// TIA Portal project "ASANSÖÖÖÖÖÖÖR" (V16)

(* hardware
DEVICE "S7-1200 station_1"  S7-1200 Station
   slot 0: "Rack_0"  S7-1200 Rack  Rack  V1.0
   slot 1: "PLC_1"  CPU 1212C DC/DC/Rly  6ES7 212-1HE40-0XB0  V4.4
*)

// ===== PLC "PLC_1"  CPU 1212C DC/DC/Rly =====

VAR_GLOBAL   // PLC tag table "Default tag table"
   "Kat 1 set yukarı" AT %M0.0 : Bool;
   "Kat 3 start" AT %I0.2 : Bool;
   "Kat 2 start" AT %I0.1 : Bool;
   "Set 3" AT %M0.2 : Bool;
   "Sensör 2" AT %I0.0 : Bool;
   "Kat 2 set yukarı" AT %M0.1 : Bool;
   "Kat 1 start" AT %I0.4 : Bool;
   "Sensör 1" AT %I0.5 : Bool;
   "Kat 2 aşağı" AT %M0.4 : Bool;
   "Kat 3 start set" AT %Q0.3 : Bool;
   "Kat 2 start set" AT %Q0.4 : Bool;
   "Kat 1 start set" AT %Q0.5 : Bool;
   "Sensör 3" AT %I0.6 : Bool;
   "Motor Yukarı" AT %Q0.2 : Bool;
   "Motor aşağı" AT %Q0.1 : Bool;
   "Kat 3 aşağı" AT %M0.3 : Bool;
END_VAR

ORGANIZATION_BLOCK "Main"   // OB1, LAD, ProgramCycle
TITLE = "Main Program Sweep (Cycle)"
{ S7_Optimized_Access := 'TRUE' }
VERSION : 0.1
   VAR_INPUT
      Initial_Call : Bool;   // Initial call of this OB
      Remanence : Bool;   // =True, if remanent data are available
   END_VAR
BEGIN

REGION Network 1
   // Kat 1 yukarı
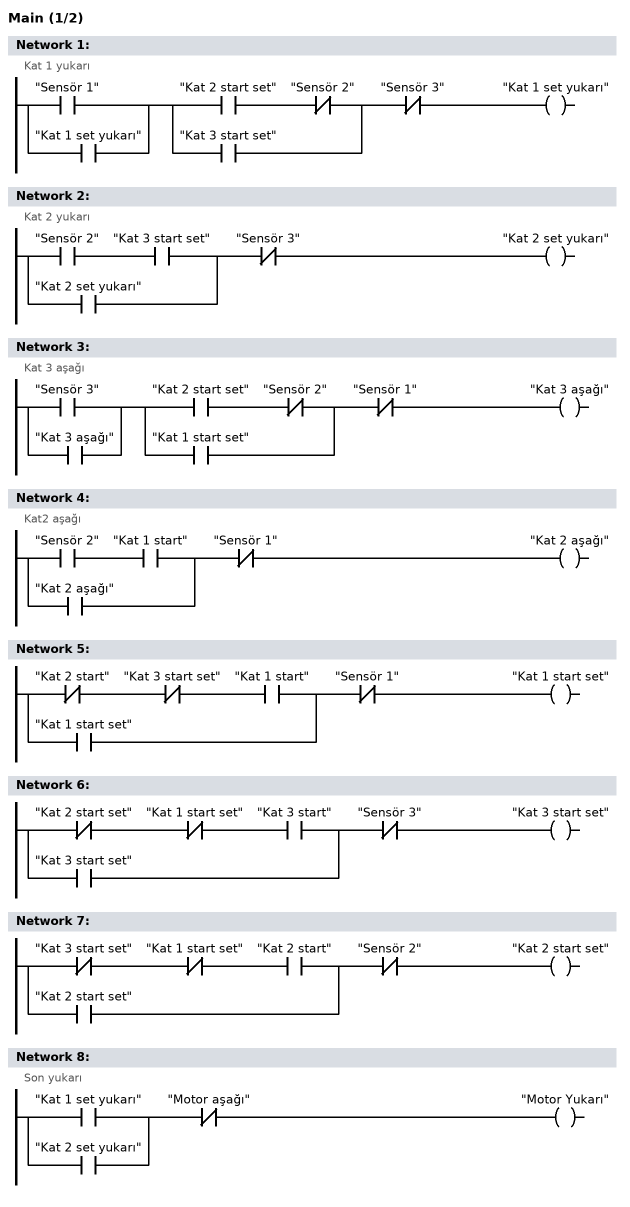
   RUNG wire#powerrail
      Contact( "Sensör 1" )
      wire#w1
      Contact( "Kat 2 start set" )
      I_Contact( "Sensör 2" )
      wire#w2
      I_Contact( "Sensör 3" )
      Coil( "Kat 1 set yukarı" )
   END_RUNG
   RUNG wire#powerrail
      Contact( "Kat 1 set yukarı" )
   END_RUNG wire#w1
   RUNG wire#w1
      Contact( "Kat 3 start set" )
   END_RUNG wire#w2
   // the same network as SCL:
   "Kat 1 set yukarı" := ("Sensör 1" OR "Kat 1 set yukarı") AND (("Kat 2 start set" AND NOT "Sensör 2") OR "Kat 3 start set") AND NOT "Sensör 3";
END_REGION

REGION Network 2
   // Kat 2 yukarı
   RUNG wire#powerrail
      Contact( "Sensör 2" )
      Contact( "Kat 3 start set" )
      wire#w1
      I_Contact( "Sensör 3" )
      Coil( "Kat 2 set yukarı" )
   END_RUNG
   RUNG wire#powerrail
      Contact( "Kat 2 set yukarı" )
   END_RUNG wire#w1
   // the same network as SCL:
   "Kat 2 set yukarı" := (("Sensör 2" AND "Kat 3 start set") OR "Kat 2 set yukarı") AND NOT "Sensör 3";
END_REGION

REGION Network 3
   // Kat 3 aşağı
   RUNG wire#powerrail
      Contact( "Sensör 3" )
      wire#w1
      Contact( "Kat 2 start set" )
      I_Contact( "Sensör 2" )
      wire#w2
      I_Contact( "Sensör 1" )
      Coil( "Kat 3 aşağı" )
   END_RUNG
   RUNG wire#powerrail
      Contact( "Kat 3 aşağı" )
   END_RUNG wire#w1
   RUNG wire#w1
      Contact( "Kat 1 start set" )
   END_RUNG wire#w2
   // the same network as SCL:
   "Kat 3 aşağı" := ("Sensör 3" OR "Kat 3 aşağı") AND (("Kat 2 start set" AND NOT "Sensör 2") OR "Kat 1 start set") AND NOT "Sensör 1";
END_REGION

REGION Network 4
   // Kat2 aşağı
   RUNG wire#powerrail
      Contact( "Sensör 2" )
      Contact( "Kat 1 start" )
      wire#w1
      I_Contact( "Sensör 1" )
      Coil( "Kat 2 aşağı" )
   END_RUNG
   RUNG wire#powerrail
      Contact( "Kat 2 aşağı" )
   END_RUNG wire#w1
   // the same network as SCL:
   "Kat 2 aşağı" := (("Sensör 2" AND "Kat 1 start") OR "Kat 2 aşağı") AND NOT "Sensör 1";
END_REGION

REGION Network 5
   RUNG wire#powerrail
      I_Contact( "Kat 2 start" )
      I_Contact( "Kat 3 start set" )
      Contact( "Kat 1 start" )
      wire#w1
      I_Contact( "Sensör 1" )
      Coil( "Kat 1 start set" )
   END_RUNG
   RUNG wire#powerrail
      Contact( "Kat 1 start set" )
   END_RUNG wire#w1
   // the same network as SCL:
   "Kat 1 start set" := ((NOT "Kat 2 start" AND NOT "Kat 3 start set" AND "Kat 1 start") OR "Kat 1 start set") AND NOT "Sensör 1";
END_REGION

REGION Network 6
   RUNG wire#powerrail
      I_Contact( "Kat 2 start set" )
      I_Contact( "Kat 1 start set" )
      Contact( "Kat 3 start" )
      wire#w1
      I_Contact( "Sensör 3" )
      Coil( "Kat 3 start set" )
   END_RUNG
   RUNG wire#powerrail
      Contact( "Kat 3 start set" )
   END_RUNG wire#w1
   // the same network as SCL:
   "Kat 3 start set" := ((NOT "Kat 2 start set" AND NOT "Kat 1 start set" AND "Kat 3 start") OR "Kat 3 start set") AND NOT "Sensör 3";
END_REGION

REGION Network 7
   RUNG wire#powerrail
      I_Contact( "Kat 3 start set" )
      I_Contact( "Kat 1 start set" )
      Contact( "Kat 2 start" )
      wire#w1
      I_Contact( "Sensör 2" )
      Coil( "Kat 2 start set" )
   END_RUNG
   RUNG wire#powerrail
      Contact( "Kat 2 start set" )
   END_RUNG wire#w1
   // the same network as SCL:
   "Kat 2 start set" := ((NOT "Kat 3 start set" AND NOT "Kat 1 start set" AND "Kat 2 start") OR "Kat 2 start set") AND NOT "Sensör 2";
END_REGION

REGION Network 8
   // Son yukarı
   RUNG wire#powerrail
      Contact( "Kat 1 set yukarı" )
      wire#w1
      I_Contact( "Motor aşağı" )
      Coil( "Motor Yukarı" )
   END_RUNG
   RUNG wire#powerrail
      Contact( "Kat 2 set yukarı" )
   END_RUNG wire#w1
   // the same network as SCL:
   "Motor Yukarı" := ("Kat 1 set yukarı" OR "Kat 2 set yukarı") AND NOT "Motor aşağı";
END_REGION

REGION Network 9: Son aşağı
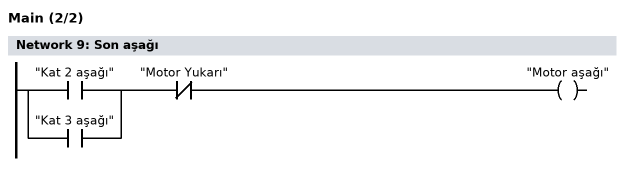
   RUNG wire#powerrail
      Contact( "Kat 2 aşağı" )
      wire#w1
      I_Contact( "Motor Yukarı" )
      Coil( "Motor aşağı" )
   END_RUNG
   RUNG wire#powerrail
      Contact( "Kat 3 aşağı" )
   END_RUNG wire#w1
   // the same network as SCL:
   "Motor aşağı" := ("Kat 2 aşağı" OR "Kat 3 aşağı") AND NOT "Motor Yukarı";
END_REGION
END_ORGANIZATION_BLOCK